// TIA Portal V19 export
TYPE "LAF_typeSR1000Parameters"
// stored: Access Published
   STRUCT
      referenceDesignator : String[20];
      simActive : Bool;   // Manual mode parameters for axis control interface
      simError : Int;
      preRescanCounter : Int;
      hwd : HW_ANY;
      telegram : "LEXCHANGETRAY_typeSr1000ProfinetTelegram";
   END_STRUCT;
END_TYPE
